FUNCTION_BLOCK StepTimeOutTimer
VAR_IN_OUT
	step : INT;
END_VAR
VAR_INPUT
	TimeOut : TIME := T#30S;
END_VAR
VAR_OUTPUT
	hasTimeOut : BOOL;
END_VAR
VAR
	Timer : TON;
	oldStep : INT;
END_VAR

Timer(IN := oldStep = step, PT := TimeOut);
IF Timer.Q THEN
	hasTimeOut := TRUE;
ELSE
	hasTimeOut := FALSE;
END_IF
oldStep := step;

END_FUNCTION_BLOCK

(* stored: Version 1.1.0.1, ProductVersion 3.1.4024.12
   POU StepTimeOutTimer: Id {d4de079f-07ca-44b1-9d08-dc0e965eeb4c}, SpecialFunc None *)
